Universal Robots PolyScope program: Main2.urp

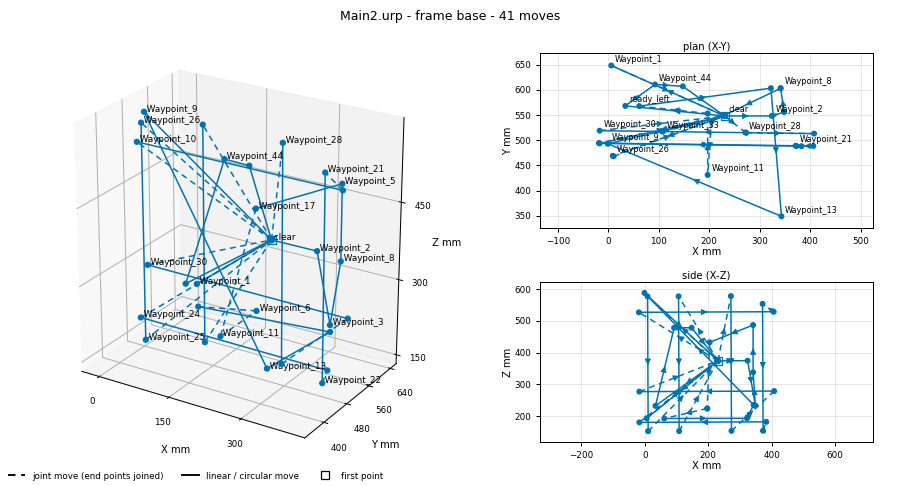
[picture p0: tool path of Main2.urp in frame base, 41 of 41 moves have a stored position in this frame; points joined in program order, loops and branches not executed]
Program Main2 (installation=main2 directory=/programs/new folder createdIn=5.11.5.1010327 lastSavedIn=5.11.5.1010327 robotSerialNumber=20215500677)
Calibrated DH parameters: a=[0.000204, -0.239222, -0.391845, -0.000001, 0.000022, 0]; d=[0.162722, -355.808559, 353.37206, 2.570385, 0.099741, 0.099629]; alpha=[1.571124, 0.000988, 0.008295, 1.568963, -1.570303, 0]; deltaTheta=[0, -0.973091, 7.204745, 0.05153, 0, 0]
Robot Program (runOnlyOnce=true)
  MoveJ speed 60 deg/s, acceleration 80 deg/s^2 (useActiveTCP=false positionType=JointAngles) tcp=DynabradeDual; feature=CubeFront
    Waypoint clear: TCP in base x=230.665 y=548.148 z=374.028 mm, rx=-1.581 ry=-0.1157 rz=-0.0213 rad; joints [213.936, -93.222, 128.559, -101.069, 49.98, -131.767] deg; TCP offset x=3.18 y=114.64 z=98.2 mm, rx=-0.7854 ry=0 rz=0 rad; feature pose in base x=9.685 y=618.378 z=176.869 mm, rx=1.5687 ry=-0.014 rz=-0.0074 rad
    URCap Zero FT Sensor (Robotiq_Copilot, Robotiq Inc.) dataModel(NodeInitializedKey=true, WaitForSteadyWrenchOptionKey=true)
  Folder sandFront
    MoveJ speed 60 deg/s, acceleration 80 deg/s^2 (useActiveTCP=false positionType=JointAngles) tcp=DynabradeDual; feature=CubeFront
      Waypoint clear: TCP in base x=230.665 y=548.148 z=374.028 mm, rx=-1.581 ry=-0.1157 rz=-0.0213 rad; joints [213.936, -93.222, 128.559, -101.069, 49.98, -131.767] deg
    MoveL speed 250 mm/s, acceleration 1200 mm/s^2 (useActiveTCP=false) tcp=DynabradeDual; feature=CubeFront
      Waypoint Waypoint_1: TCP in base x=6.072 y=648.1 z=192.982 mm, rx=-1.5699 ry=0.0092 rz=0.0097 rad; joints [251.403, -67.593, 131.535, -110.394, 77.851, -166.352] deg; feature pose in base x=6.058 y=653.089 z=192.929 mm, rx=1.5716 ry=0.003 rz=-0.0025 rad
      URCap Finishing Tool Control (Robotiq_Copilot, Robotiq Inc.) dataModel(ToolOutputNameKey=digital_out[0], HackTriggeringContributionIsDefinedMethodKey=true)
      URCap Zero FT Sensor (Robotiq_Copilot, Robotiq Inc.) dataModel(NodeInitializedKey=true, WaitForSteadyWrenchOptionKey=true)
      Wait Sleep waitTime=2
      URCap Find Surface (Robotiq_Copilot, Robotiq Inc.) dataModel(NodeInitializedKey=true, WaitForSteadyWrenchOptionKey=false, ls_force=10.0, ls_distance=100.0, ls_speed=5.0, ZeroSensorBeforeKey=true, ls_if_distance=false, ls_if_force=false); state(isChildrenLocked=true)
        'Add Stop conditions from the Find Surface node'
    MoveL speed 60 mm/s, acceleration 1200 mm/s^2 (useActiveTCP=false) tcp=DynabradeDual; feature=CubeFront
      Force Simple feature=Joint_6_name; selection=[0, 0, 1, 0, 0, 0]; wrench=[0, 0, 5, 0, 0, 0]; limitsForce=[0.15, 0.15, 0.15, 1.047198, 1.047198, 1.047198]; limitsMotion=[0.1, 0.1, 0.1, 0.349066, 0.349066, 0.349066]
        MoveDirectionNode (selectedDirection=YPlus) feature(featureName=CubeFront)
          Until DISTANCE (allowActions=false deceleration=3 distanceNodeType=STOP) Distance=0.355; motionParameters(blendRadius=0)
        MoveDirectionNode (selectedDirection=XPlus) feature(featureName=CubeFront)
          Until DISTANCE (allowActions=false deceleration=3 distanceNodeType=STOP) Distance=0.355; motionParameters(blendRadius=0)
        MoveDirectionNode (selectedDirection=YMinus) feature(featureName=CubeFront)
          Until DISTANCE (allowActions=false deceleration=3 distanceNodeType=STOP) Distance=0.355; motionParameters(blendRadius=0)
        MoveDirectionNode (selectedDirection=XMinus) feature(featureName=CubeFront)
          Until DISTANCE (allowActions=false deceleration=3 distanceNodeType=STOP) Distance=0.355; motionParameters(blendRadius=0)
        URCap Finishing Tool Control (Robotiq_Copilot, Robotiq Inc.) dataModel(FinishingToolStateKey=false, ToolOutputNameKey=digital_out[0], HackTriggeringContributionIsDefinedMethodKey=true)
      MoveDirectionNode (selectedDirection=ZMinus) feature=Joint_6_name
        Until DISTANCE (allowActions=false deceleration=3 distanceNodeType=STOP) Distance=0.025; motionParameters(blendRadius=0)
    MoveJ speed 60 deg/s, acceleration 80 deg/s^2 (useActiveTCP=true positionType=JointAngles) feature=Base
      Waypoint clear: TCP in base x=230.665 y=548.148 z=374.028 mm, rx=-1.581 ry=-0.1157 rz=-0.0213 rad; joints [213.936, -93.222, 128.559, -101.069, 49.98, -131.767] deg; feature pose in base x=9.685 y=618.378 z=176.869 mm, rx=1.5687 ry=-0.014 rz=-0.0074 rad
  Folder sandRebate
    MoveJ speed 60 deg/s, acceleration 80 deg/s^2 (useActiveTCP=false) tcp=DynabradeDual; feature=CubeFront
      Waypoint clear: TCP in base x=230.665 y=548.148 z=374.028 mm, rx=-1.581 ry=-0.1157 rz=-0.0213 rad; joints [213.936, -93.222, 128.559, -101.069, 49.98, -131.767] deg
      URCap Zero FT Sensor (Robotiq_Copilot, Robotiq Inc.) dataModel(NodeInitializedKey=true, WaitForSteadyWrenchOptionKey=true)
      MoveL speed 250 mm/s, acceleration 1200 mm/s^2 (useActiveTCP=false) tcp=DynabradeDual; feature=CubeFront
        Waypoint ready_left: TCP in base x=33.773 y=568.14 z=232.075 mm, rx=-1.2213 ry=-1.2022 rz=1.1979 rad; joints [233.005, -43.676, 101.374, -178.142, 55.004, -44.435] deg; TCP offset x=3.18 y=114.64 z=98.2 mm, rx=-0.7854 ry=0 rz=0 rad
        URCap Find Surface (Robotiq_Copilot, Robotiq Inc.) dataModel(NodeInitializedKey=true, WaitForSteadyWrenchOptionKey=false, ls_force=10.0, ls_distance=100.0, ls_speed=5.0, ZeroSensorBeforeKey=true, ls_if_distance=false, ls_if_force=false); state(isChildrenLocked=true)
          'Add Stop conditions from the Find Surface node'
        URCap Finishing Tool Control (Robotiq_Copilot, Robotiq Inc.) dataModel(ToolOutputNameKey=digital_out[0], HackTriggeringContributionIsDefinedMethodKey=true)
        Wait Sleep waitTime=0.5
        Force Simple feature=Joint_6_name; selection=[0, 0, 1, 0, 0, 0]; wrench=[0, 0, 3, 0, 0, 0]; limitsForce=[0.15, 0.15, 0.15, 1.047198, 1.047198, 1.047198]; limitsMotion=[0.1, 0.1, 0.1, 0.349066, 0.349066, 0.349066]
          Waypoint Waypoint_44: motionParameters(jointSpeed=1.047198 jointAcceleration=1.396263 cartesianSpeed=0.05 cartesianAcceleration=1.2); TCP in base x=92.634 y=610.628 z=478.238 mm, rx=-0.8396 ry=-1.4025 rz=0.8393 rad; joints [232.816, -51.553, 73.036, -159.375, 69.035, -55.707] deg; TCP offset x=3.18 y=114.64 z=98.2 mm, rx=-0.7854 ry=0 rz=0 rad; feature pose in base x=85.344 y=655.608 z=190.328 mm, rx=1.5707 ry=0.001 rz=-0.0012 rad
        URCap Finishing Tool Control (Robotiq_Copilot, Robotiq Inc.) dataModel(ToolOutputNameKey=digital_out[0], HackTriggeringContributionIsDefinedMethodKey=true, FinishingToolStateKey=false)
        Waypoint Waypoint_4: TCP in base x=147.72 y=606.874 z=478.224 mm, rx=-0.8396 ry=-1.4025 rz=0.8394 rad; joints [229.161, -48.232, 67.407, -157.963, 71.791, -53.121] deg
        Waypoint clear: TCP in base x=230.665 y=548.148 z=374.028 mm, rx=-1.581 ry=-0.1157 rz=-0.0213 rad; joints [213.936, -93.222, 128.559, -101.069, 49.98, -131.767] deg; feature pose in base x=9.685 y=618.378 z=176.869 mm, rx=1.5687 ry=-0.014 rz=-0.0074 rad
        Waypoint Waypoint_2: TCP in base x=324.212 y=548.214 z=374.491 mm, rx=-1.2092 ry=1.2092 rz=-1.2092 rad; joints [245.591, -72.937, 106.11, -100.873, 130.52, -237.51] deg; feature pose in base x=6.058 y=653.089 z=192.929 mm, rx=1.5716 ry=0.003 rz=-0.0025 rad
        Waypoint Waypoint_3: TCP in base x=348.632 y=555.868 z=233.406 mm, rx=-1.199 ry=1.2125 rz=-1.2251 rad; joints [243.702, -57.561, 109.561, -119.163, 129.636, -236.605] deg; TCP offset x=3.18 y=114.64 z=98.2 mm, rx=-0.7854 ry=0 rz=0 rad; feature pose in base x=9.685 y=618.378 z=176.869 mm, rx=1.5687 ry=-0.014 rz=-0.0074 rad
        URCap Zero FT Sensor (Robotiq_Copilot, Robotiq Inc.) dataModel(NodeInitializedKey=true, WaitForSteadyWrenchOptionKey=true)
        URCap Find Surface (Robotiq_Copilot, Robotiq Inc.) dataModel(NodeInitializedKey=true, WaitForSteadyWrenchOptionKey=false, ls_force=10.0, ls_distance=100.0, ls_speed=5.0, ZeroSensorBeforeKey=true, ls_if_distance=false, ls_if_force=false); state(isChildrenLocked=true)
          'Add Stop conditions from the Find Surface node'
        URCap Finishing Tool Control (Robotiq_Copilot, Robotiq Inc.) dataModel(ToolOutputNameKey=digital_out[0], HackTriggeringContributionIsDefinedMethodKey=true)
        Wait Sleep waitTime=0.5
        Force Simple feature=Joint_6_name; selection=[0, 0, 1, 0, 0, 0]; wrench=[0, 0, 3, 0, 0, 0]; limitsForce=[0.15, 0.15, 0.15, 1.047198, 1.047198, 1.047198]; limitsMotion=[0.1, 0.1, 0.1, 0.349066, 0.349066, 0.349066]
          Waypoint Waypoint_8: motionParameters(jointSpeed=1.047198 jointAcceleration=1.396263 cartesianSpeed=0.05 cartesianAcceleration=1.2); TCP in base x=341.551 y=603.074 z=337.804 mm, rx=-2.2214 ry=0 rz=-2.2214 rad; joints [243.714, -66.77, 84.264, -17.409, 108.783, -269.646] deg; TCP offset x=3.18 y=114.64 z=98.2 mm, rx=-0.7854 ry=0 rz=0 rad; feature pose in base x=6.058 y=653.089 z=192.929 mm, rx=1.5716 ry=0.003 rz=-0.0025 rad
          Waypoint Waypoint_5: motionParameters(jointSpeed=1.047198 jointAcceleration=1.396263 cartesianSpeed=0.05 cartesianAcceleration=1.2); TCP in base x=341.546 y=602.951 z=486.88 mm, rx=2.115 ry=0.2149 rz=2.1148 rad; joints [243.737, -66.909, 60.838, 14.812, 108.93, -275.062] deg; TCP offset x=3.18 y=114.64 z=98.2 mm, rx=-0.7854 ry=0 rz=0 rad
        URCap Finishing Tool Control (Robotiq_Copilot, Robotiq Inc.) dataModel(FinishingToolStateKey=false, ToolOutputNameKey=digital_out[0], HackTriggeringContributionIsDefinedMethodKey=true)
        Waypoint Waypoint_17: TCP in base x=204.615 y=537.314 z=432.533 mm, rx=-1.1836 ry=-1.1482 rz=-1.3158 rad; joints [212.134, -87.867, 98.846, 1.992, -9.504, -287.219] deg; TCP offset x=3.18 y=114.64 z=98.2 mm, rx=-0.7854 ry=0 rz=0 rad
        MoveJ speed 60 deg/s, acceleration 80 deg/s^2 (useActiveTCP=true) feature=CubeFront
          Waypoint Waypoint_11: TCP in base x=197.023 y=431.256 z=223.624 mm, rx=2.362 ry=2.0713 rz=0 rad; joints [223.025, -89.028, 102.064, -70.501, -56.519, -139.472] deg
          Waypoint Waypoint_6: TCP in base x=196.959 y=553.123 z=223.756 mm, rx=-1.75 ry=-2.609 rz=-0.0001 rad; joints [233.913, -69.804, 77.285, -56.958, -67.897, -156.703] deg
          Waypoint Waypoint_31: TCP in base x=61.467 y=567.687 z=192.19 mm, rx=1.7638 ry=2.5902 rz=0.0029 rad; joints [245.976, -73.297, 87.687, -68.963, -60.284, -145.062] deg; TCP offset x=3.18 y=114.64 z=98.2 mm, rx=-0.7854 ry=0 rz=0 rad; feature pose in base x=9.685 y=618.378 z=176.869 mm, rx=1.5687 ry=-0.014 rz=-0.0074 rad
          URCap Zero FT Sensor (Robotiq_Copilot, Robotiq Inc.) dataModel(NodeInitializedKey=true, WaitForSteadyWrenchOptionKey=true)
        URCap Find Surface (Robotiq_Copilot, Robotiq Inc.) dataModel(NodeInitializedKey=true, ZeroSensorBeforeKey=true, WaitForSteadyWrenchOptionKey=false, ls_force=10.0, ls_distance=100.0, ls_speed=5.0, ls_if_distance=false, ls_if_force=false); state(isChildrenLocked=true)
          'Add Stop conditions from the Find Surface node'
        URCap Finishing Tool Control (Robotiq_Copilot, Robotiq Inc.) dataModel(ToolOutputNameKey=digital_out[0], HackTriggeringContributionIsDefinedMethodKey=true)
        Wait Sleep waitTime=0.5
        Force Simple feature=Joint_6_name; selection=[0, 0, 1, 0, 0, 0]; wrench=[0, 0, 1, 0, 0, 0]; limitsForce=[0.15, 0.15, 0.15, 1.047198, 1.047198, 1.047198]; limitsMotion=[0.1, 0.1, 0.1, 0.349066, 0.349066, 0.349066]
          Waypoint Waypoint_7: motionParameters(jointSpeed=1.047198 jointAcceleration=1.396263 cartesianSpeed=0.05 cartesianAcceleration=1.2); TCP in base x=322.305 y=603.203 z=193.01 mm, rx=2.5491 ry=1.8349 rz=-0.0035 rad; joints [225.958, -61.111, 72.887, -78.246, -49.944, -124.133] deg; TCP offset x=3.18 y=114.64 z=98.2 mm, rx=-0.7854 ry=0 rz=0 rad; feature pose in base x=6.058 y=653.089 z=192.929 mm, rx=1.5716 ry=0.003 rz=-0.0025 rad
        URCap Finishing Tool Control (Robotiq_Copilot, Robotiq Inc.) dataModel(FinishingToolStateKey=false, ToolOutputNameKey=digital_out[0], HackTriggeringContributionIsDefinedMethodKey=true)
        Waypoint Waypoint_13: TCP in base x=343.245 y=349.195 z=234.967 mm, rx=-1.8514 ry=-2.5381 rz=0.0001 rad; joints [208.052, -81.166, 89.339, -53.576, -82.434, -172.912] deg; feature pose in base x=9.685 y=618.378 z=176.869 mm, rx=1.5687 ry=-0.014 rz=-0.0074 rad
        Waypoint Waypoint_9: TCP in base x=-0.811 y=492.962 z=588.061 mm, rx=-1.9827 ry=-0.1778 rz=-0.0774 rad; joints [237.765, -113.533, 89.133, -2.101, 52.621, -171.272] deg
        Waypoint clear: TCP in base x=230.665 y=548.148 z=374.028 mm, rx=-1.581 ry=-0.1157 rz=-0.0213 rad; joints [213.936, -93.222, 128.559, -101.069, 49.98, -131.767] deg; feature pose in base x=9.685 y=618.378 z=176.869 mm, rx=1.5687 ry=-0.014 rz=-0.0074 rad
  SuppressedNode
    Folder Chamfer
      MoveL speed 250 mm/s, acceleration 1200 mm/s^2 (useActiveTCP=true) feature=Base
        MoveJ speed 60 deg/s, acceleration 80 deg/s^2 (useActiveTCP=true) feature=CubeFront
          Waypoint Waypoint_14: TCP in base x=40.557 y=344.633 z=644.318 mm, rx=1.3155 ry=-1.3725 rz=-1.2523 rad; joints [213.145, -95.792, 65.461, -31.373, -65.462, -328.995] deg; feature pose in base x=6.058 y=653.089 z=192.929 mm, rx=1.5716 ry=0.003 rz=-0.0025 rad
          Waypoint Waypoint_15: TCP in base x=-6.602 y=417.802 z=666.352 mm, rx=-2.8064 ry=0.3635 rz=0.257 rad; joints [242.083, -106.85, 75.59, -118.753, -70.655, -356.384] deg
          Waypoint Waypoint_16: TCP in base x=7.321 y=653.157 z=552.583 mm, rx=-2.3553 ry=0.0014 rz=0.0042 rad; joints [252.243, -84.14, 86.654, -182.715, -72.191, -359.211] deg
        URCap Find Surface (Robotiq_Copilot, Robotiq Inc.) dataModel(NodeInitializedKey=true, ZeroSensorBeforeKey=true, WaitForSteadyWrenchOptionKey=false, ls_force=10.0, ls_distance=100.0, ls_speed=5.0, ls_if_distance=false, ls_if_force=false); state(isChildrenLocked=true)
          'Add Stop conditions from the Find Surface node'
        URCap Finishing Tool Control (Robotiq_Copilot, Robotiq Inc.) dataModel(ToolOutputNameKey=digital_out[0], HackTriggeringContributionIsDefinedMethodKey=true)
        Wait Sleep waitTime=0.5
        MoveDirectionNode (selectedDirection=XPlus toolParams=0.15, 1.2) feature(featureName=CubeFront)
          Until DISTANCE (allowActions=false deceleration=3 distanceNodeType=STOP) Distance=0.35; motionParameters(blendRadius=0)
        MoveDirectionNode (selectedDirection=ZMinus) feature=Joint_6_name
          Until DISTANCE (allowActions=false deceleration=3 distanceNodeType=STOP) Distance=0.025; motionParameters(blendRadius=0)
        URCap Finishing Tool Control (Robotiq_Copilot, Robotiq Inc.) dataModel(FinishingToolStateKey=false, ToolOutputNameKey=digital_out[0], HackTriggeringContributionIsDefinedMethodKey=true)
        Waypoint Waypoint_18: TCP in base x=366.179 y=605.982 z=520.828 mm, rx=-1.6861 ry=0.1385 rz=1.2496 rad; joints [208.374, -44.818, 51.064, -237.69, -37.068, -253.683] deg
        URCap Find Surface (Robotiq_Copilot, Robotiq Inc.) dataModel(NodeInitializedKey=true, ZeroSensorBeforeKey=true, WaitForSteadyWrenchOptionKey=false, ls_force=10.0, ls_distance=100.0, ls_speed=5.0, ls_if_distance=false, ls_if_force=false); state(isChildrenLocked=true)
          'Add Stop conditions from the Find Surface node'
        URCap Finishing Tool Control (Robotiq_Copilot, Robotiq Inc.) dataModel(ToolOutputNameKey=digital_out[0], HackTriggeringContributionIsDefinedMethodKey=true)
        MoveDirectionNode (selectedDirection=YMinus toolParams=0.15, 1.2) feature(featureName=CubeFront)
          Until DISTANCE (allowActions=false deceleration=3 distanceNodeType=STOP) Distance=0.35; motionParameters(blendRadius=0)
        URCap Finishing Tool Control (Robotiq_Copilot, Robotiq Inc.) dataModel(FinishingToolStateKey=false, ToolOutputNameKey=digital_out[0], HackTriggeringContributionIsDefinedMethodKey=true)
        MoveDirectionNode (selectedDirection=ZMinus) feature=Joint_6_name
          Until DISTANCE (allowActions=false deceleration=3 distanceNodeType=STOP) Distance=0.05; motionParameters(blendRadius=0)
        Waypoint Waypoint_20: TCP in base x=366.722 y=626.869 z=194.22 mm, rx=-1.1174 ry=-0.6786 rz=-0.9417 rad; joints [212.764, -30.352, 68.609, -330.279, -35.41, -327.866] deg
        URCap Find Surface (Robotiq_Copilot, Robotiq Inc.) dataModel(NodeInitializedKey=true, ZeroSensorBeforeKey=true, WaitForSteadyWrenchOptionKey=false, ls_force=10.0, ls_distance=100.0, ls_speed=5.0, ls_if_distance=false, ls_if_force=false); state(isChildrenLocked=true)
          'Add Stop conditions from the Find Surface node'
        URCap Finishing Tool Control (Robotiq_Copilot, Robotiq Inc.) dataModel(ToolOutputNameKey=digital_out[0], HackTriggeringContributionIsDefinedMethodKey=true)
        Waypoint Waypoint_19: motionParameters(jointSpeed=1.047198 jointAcceleration=1.396263 cartesianSpeed=0.05 cartesianAcceleration=1.2); TCP in base x=29.784 y=640.794 z=212.679 mm, rx=-1.2502 ry=-0.1072 rz=-0.0765 rad; joints [247.483, -34.268, 98.117, -310.948, -74.468, -342.493] deg
        URCap Finishing Tool Control (Robotiq_Copilot, Robotiq Inc.) dataModel(FinishingToolStateKey=false, ToolOutputNameKey=digital_out[0], HackTriggeringContributionIsDefinedMethodKey=true)
        MoveDirectionNode (selectedDirection=ZMinus) feature=Joint_6_name
          Until DISTANCE (allowActions=false deceleration=3 distanceNodeType=STOP) Distance=0.05; motionParameters(blendRadius=0)
  Folder SprayFront
    MoveJ speed 60 deg/s, acceleration 80 deg/s^2 (useActiveTCP=false) tcp=DynabradeDual; feature=CubeFront
      Waypoint clear: TCP in base x=230.665 y=548.148 z=374.028 mm, rx=-1.581 ry=-0.1157 rz=-0.0213 rad; joints [213.936, -93.222, 128.559, -101.069, 49.98, -131.767] deg; feature pose in base x=9.685 y=618.378 z=176.869 mm, rx=1.5687 ry=-0.014 rz=-0.0074 rad
    MoveJ speed 60 deg/s, acceleration 80 deg/s^2 (useActiveTCP=false) tcp=Spray; feature=CubeFront
      Waypoint Waypoint_10: TCP in base x=-18.468 y=494.451 z=527.007 mm, rx=-0.0631 ry=2.1556 rz=2.1464 rad; joints [251.333, -72.134, 115.852, 89.334, -71.596, -348.276] deg; TCP offset x=20.839 y=-27.14 z=105.994 mm, rx=0.1226 ry=1.1769 rz=2.8697 rad
      Call StartSpray
    MoveL speed 100 mm/s, acceleration 1200 mm/s^2 (useActiveTCP=true) feature=CubeFront
      Waypoint Waypoint_12: TCP in base x=406.466 y=488.644 z=528.84 mm, rx=-0.0631 ry=2.1554 rz=2.1465 rad; joints [207.201, -51.632, 76.045, 84.569, -47.479, -304.205] deg; TCP offset x=20.839 y=-27.14 z=105.994 mm, rx=0.1226 ry=1.1769 rz=2.8697 rad
      Call stopSpray
    MoveJ speed 60 deg/s, acceleration 80 deg/s^2 (useActiveTCP=false) tcp=Spray; feature=CubeFront
      Waypoint Waypoint_21: TCP in base x=371.408 y=489.224 z=553.631 mm, rx=-1.2033 ry=1.1607 rz=1.1716 rad; joints [201.954, -55.469, 35.436, 9.234, -22.213, -259.505] deg
      Call StartSpray
    MoveL speed 100 mm/s, acceleration 1200 mm/s^2 (useActiveTCP=false) tcp=Spray; feature=CubeFront
      Waypoint Waypoint_22: TCP in base x=373.023 y=488.37 z=153.653 mm, rx=-1.2033 ry=1.1607 rz=1.1716 rad; joints [201.811, -46.917, 82.081, -46.163, -21.934, -259.291] deg
      Call stopSpray
    MoveJ speed 60 deg/s, acceleration 80 deg/s^2 (useActiveTCP=false) tcp=Spray; feature=CubeFront
      Waypoint Waypoint_23: TCP in base x=382.922 y=488.301 z=181.714 mm, rx=0.0103 ry=2.2147 rz=2.2103 rad; joints [209.131, -21.562, 81.485, 53.437, -50.089, -303.679] deg
      Call StartSpray
    MoveL speed 100 mm/s, acceleration 1200 mm/s^2 (useActiveTCP=false) tcp=Spray; feature=CubeFront
      Waypoint Waypoint_24: TCP in base x=-17.013 y=493.762 z=180.055 mm, rx=0.0103 ry=2.2147 rz=2.2103 rad; joints [253.121, -24.563, 110.523, 47.647, -75.487, -344.997] deg
      Call stopSpray
    MoveJ speed 60 deg/s, acceleration 80 deg/s^2 (useActiveTCP=false positionType=JointAngles) tcp=Spray; feature=CubeFront
      Waypoint clear: TCP in base x=230.665 y=548.148 z=374.028 mm, rx=-1.581 ry=-0.1157 rz=-0.0213 rad; joints [213.936, -93.222, 128.559, -101.069, 49.98, -131.767] deg; TCP offset x=3.18 y=114.64 z=98.2 mm, rx=-0.7854 ry=0 rz=0 rad
    MoveJ speed 60 deg/s, acceleration 80 deg/s^2 (useActiveTCP=false) tcp=Spray; feature=CubeFront
      Waypoint Waypoint_26: TCP in base x=8.963 y=469.193 z=577.186 mm, rx=-1.2027 ry=1.214 rz=1.1952 rad; joints [222.592, -107.476, 101.75, -61.506, -3.487, -199.197] deg; TCP offset x=20.839 y=-27.14 z=105.994 mm, rx=0.1226 ry=1.1769 rz=2.8697 rad
      Call StartSpray
    MoveL speed 100 mm/s, acceleration 1200 mm/s^2 (useActiveTCP=false) tcp=Spray; feature=CubeFront
      Waypoint Waypoint_25: TCP in base x=10.718 y=468.315 z=152.199 mm, rx=-1.2027 ry=1.2139 rz=1.1952 rad; joints [222.113, -68.068, 142.774, -143.838, -3.758, -197.295] deg
      Call stopSpray
    MoveJ speed 60 deg/s, acceleration 80 deg/s^2 (useActiveTCP=false positionType=JointAngles) tcp=Spray; feature=CubeFront
      Waypoint clear: TCP in base x=230.665 y=548.148 z=374.028 mm, rx=-1.581 ry=-0.1157 rz=-0.0213 rad; joints [213.936, -93.222, 128.559, -101.069, 49.98, -131.767] deg; TCP offset x=3.18 y=114.64 z=98.2 mm, rx=-0.7854 ry=0 rz=0 rad
  Folder SprayRebate
    MoveJ speed 60 deg/s, acceleration 80 deg/s^2 (useActiveTCP=false positionType=JointAngles) tcp=Spray; feature=CubeFront
      Waypoint clear: TCP in base x=230.665 y=548.148 z=374.028 mm, rx=-1.581 ry=-0.1157 rz=-0.0213 rad; joints [213.936, -93.222, 128.559, -101.069, 49.98, -131.767] deg
    MoveJ speed 60 deg/s, acceleration 80 deg/s^2 (useActiveTCP=false) tcp=Spray; feature=CubeFront
      Waypoint Waypoint_28: TCP in base x=271.667 y=515.614 z=578.139 mm, rx=-0.606 ry=1.4822 rz=0.6004 rad; joints [208.011, -87.406, 104.797, -191.165, -29.317, -91.698] deg; TCP offset x=20.839 y=-27.14 z=105.994 mm, rx=0.1226 ry=1.1769 rz=2.8697 rad
      Call StartSpray
    MoveL speed 100 mm/s, acceleration 1200 mm/s^2 (useActiveTCP=false) tcp=Spray; feature=CubeFront
      Waypoint Waypoint_27: TCP in base x=273.408 y=514.734 z=153.162 mm, rx=-0.606 ry=1.4823 rz=0.6004 rad; joints [207.859, -39.21, 119.689, -253.722, -29.522, -92.302] deg
      Call stopSpray
    MoveJ speed 60 deg/s, acceleration 80 deg/s^2 (useActiveTCP=false) tcp=Spray; feature=CubeFront
      Waypoint Waypoint_29: TCP in base x=407.829 y=513.19 z=278.745 mm, rx=0.0171 ry=2.8953 rz=1.196 rad; joints [202.265, -49.904, 107.859, -237.705, -20.006, 3.393] deg; TCP offset x=20.839 y=-27.14 z=105.994 mm, rx=0.1226 ry=1.1769 rz=2.8697 rad
      Call StartSpray
    MoveL speed 100 mm/s, acceleration 1200 mm/s^2 (useActiveTCP=false) tcp=Spray; feature=CubeFront
      Waypoint Waypoint_30: TCP in base x=-17.094 y=518.98 z=276.97 mm, rx=0.0171 ry=2.8954 rz=1.196 rad; joints [250.228, -61.644, 139.534, -257.5, -68.041, 3.56] deg; TCP offset x=20.839 y=-27.14 z=105.994 mm, rx=0.1226 ry=1.1769 rz=2.8697 rad
      Call stopSpray
    MoveJ speed 60 deg/s, acceleration 80 deg/s^2 (useActiveTCP=false positionType=JointAngles) tcp=Spray; feature=CubeFront
      Waypoint clear: TCP in base x=230.665 y=548.148 z=374.028 mm, rx=-1.581 ry=-0.1157 rz=-0.0213 rad; joints [213.936, -93.222, 128.559, -101.069, 49.98, -131.767] deg; TCP offset x=3.18 y=114.64 z=98.2 mm, rx=-0.7854 ry=0 rz=0 rad
    MoveJ speed 60 deg/s, acceleration 80 deg/s^2 (useActiveTCP=false) tcp=Spray; feature=CubeFront
      Waypoint Waypoint_32: TCP in base x=106.648 y=517.867 z=577.433 mm, rx=-0.6252 ry=-1.4837 rz=-0.6245 rad; joints [231.305, -102.456, 86.054, 11.982, 51.705, -83.541] deg; TCP offset x=20.839 y=-27.14 z=105.994 mm, rx=0.1226 ry=1.1769 rz=2.8697 rad
      Call StartSpray
    MoveL speed 100 mm/s, acceleration 1200 mm/s^2 (useActiveTCP=false) tcp=Spray; feature=CubeFront
      Waypoint Waypoint_33: TCP in base x=108.397 y=516.974 z=152.506 mm, rx=-0.6252 ry=-1.4837 rz=-0.6245 rad; joints [230.83, -82.04, 136.774, -59.04, 51.734, -83.726] deg
      Call stopSpray
    MoveJ speed 60 deg/s, acceleration 80 deg/s^2 (useActiveTCP=false positionType=JointAngles) tcp=Spray; feature=CubeFront
      Waypoint clear: TCP in base x=230.665 y=548.148 z=374.028 mm, rx=-1.581 ry=-0.1157 rz=-0.0213 rad; joints [213.936, -93.222, 128.559, -101.069, 49.98, -131.767] deg; TCP offset x=3.18 y=114.64 z=98.2 mm, rx=-0.7854 ry=0 rz=0 rad
SubProgram -> StartSpray
SubProgram -> stopSpray
SubProgram StartSpray (keepSynchronizedWithDisk=false)
  Set DigitalOutput pin=digital_out[1]; digitalValue=1
  Wait Sleep waitTime=0.3
SubProgram stopSpray (keepSynchronizedWithDisk=false)
  Set DigitalOutput pin=digital_out[1]; digitalValue=0
  Wait Sleep waitTime=0.3
